(* IEC 61131-3 sources: axftcmlib/src/Axis/PosAxis, 6 files *)

(* ---- itfPosAxis.st ---- *)
USING Simatic.Ax.Commands;

NAMESPACE Simatic.Ax.axftcmlib.Motion

    INTERFACE itfPosAxis EXTENDS itfSpeedAxis

    METHOD MoveAbsolute  : itfCommand
        VAR_INPUT
            Position : LREAL; // Absolute target position
            Velocity : LReal := 100.0;
        END_VAR
    END_METHOD

    METHOD MoveRelative  : itfCommand
        VAR_INPUT
            Distance : LREAL; // Distance for the positioning process (negative or positive)
            Velocity : LReal := 100.0;
        END_VAR
    END_METHOD

    METHOD HomeDirect  : itfCommand
        VAR_INPUT
            Position : LREAL; // Distance for the positioning process (negative or positive)
        END_VAR
    END_METHOD

END_INTERFACE

END_NAMESPACE

(* ---- commandActiveHoming.st ---- *)
USING Simatic.Ax.IO.Input;
USING Simatic.Ax.IO.Input;
USING Simatic.Ax.Commands;
USING Simatic.Ax.IO.Input;

NAMESPACE Simatic.Ax.axftcmlib.Motion

    CLASS INTERNAL commandActiveHoming
        EXTENDS ExecuteCommand
        VAR
            _AxisRef : REF_TO TO_PosAxis;
            _velocity : LREAL;
            _direction : Direction;
            _position : LREAL;
            _iRefSensor : ItfBinSignal;
            _exec : BOOL;
        END_VAR

        METHOD PUBLIC Start : itfCommand
            VAR_INPUT
                AxisRef : REF_TO TO_PosAxis;
                Velocity : LREAL := 100.0;
                Direction : Direction;
                Position : LREAL := 0.0;
                RefSensor : ItfBinSignal;
            END_VAR
            _AxisRef := AxisRef;
            _velocity := Velocity;
            _direction := Direction;
            _position := Position;
            _iRefSensor := RefSensor;
            THIS.ExecuteWithRisingEdge();
            Start := THIS;
        END_METHOD

        METHOD PROTECTED OVERRIDE Execute
            IF NOT (_exec) THEN
                RETURN;
            END_IF;
            IF (NOT _AxisRef^.IsPoweredOn()) THEN
                THIS.SetError(WORD#16#8001);
            ELSE
                _AxisRef^.Run(TRUE);
                IF (_iRefSensor.QRis()) THEN
                    _AxisRef^.Run(FALSE);
                    _Done := _AxisRef^.SetPosition(value := _position);
                    ;
                END_IF;
            END_IF;
        END_METHOD

        METHOD PROTECTED OVERRIDE SetExecute
            VAR_INPUT
                exec : BOOL;
            END_VAR
            _exec := exec;
            IF (exec) THEN
                THIS.InitState();
                IF (_AxisRef = NULL) THEN
                    THIS.SetError(WORD#16#8003);
                    RETURN;
                ELSIF (_iRefSensor = NULL) THEN
                    THIS.SetError(WORD#16#8004);
                    RETURN;
                END_IF;
                IF (NOT _AxisRef^.IsPoweredOn()) THEN
                    THIS.SetError(WORD#16#8001);
                ELSIF (_AxisRef^.IsRunning()) THEN
                    THIS.SetError(WORD#16#8002); // Can not be homed because axis is not stillstanding
                END_IF;
            END_IF;
        END_METHOD
    END_CLASS

END_NAMESPACE

(* ---- commandHomeDirect.st ---- *)
USING Simatic.Ax.Commands;

NAMESPACE Simatic.Ax.axftcmlib.Motion

    CLASS INTERNAL commandHomeDirect
        EXTENDS ExecuteCommand
        VAR
            _AxisRef : REF_TO TO_PosAxis;
            _position : LReal;
        END_VAR

        METHOD PUBLIC Start : itfCommand
            VAR_INPUT
                AxisRef : REF_TO TO_PosAxis;
                Position : LREAL := 0.0;
            END_VAR
            _AxisRef := AxisRef;
            _position := Position;
            THIS.ExecuteWithRisingEdge();
            Start := THIS;
        END_METHOD

        METHOD PROTECTED OVERRIDE Execute
            IF (NOT _AxisRef^.isPowerdOn) THEN
                THIS.SetError(WORD#16#8001);
            ELSE
                ;
            END_IF;
        END_METHOD

        METHOD PROTECTED OVERRIDE SetExecute
            VAR_INPUT
                exec : BOOL;
            END_VAR
            IF (NOT _AxisRef^.isPowerdOn) THEN
                THIS.SetError(WORD#16#8001);
            ELSIF (_AxisRef^.IsRunning()) THEN
                THIS.SetError(WORD#16#8002);  // Con not be homed because axis is not stillstanding
            ELSE
                _Done := _AxisRef^.SetPosition(value := _position);
            END_IF;

        END_METHOD
    END_CLASS

END_NAMESPACE

(* ---- commandMoveAbsolute.st ---- *)
USING Simatic.Ax.Commands;

NAMESPACE Simatic.Ax.axftcmlib.Motion

    CLASS INTERNAL commandMoveAbsolute
        EXTENDS ExecuteCommand
        VAR
            _AxisRef : REF_TO TO_PosAxis;
            _velocity : LREAL;
            _position : LREAL;
        END_VAR
        VAR PRIVATE
            _execute : BOOL;
        END_VAR

        METHOD PUBLIC Start : itfCommand
            VAR_INPUT
                AxisRef : REF_TO TO_PosAxis;
                Velocity : LREAL := LREAL#100.0;
                Position : LREAL := 0.0;
            END_VAR
            _AxisRef := AxisRef;
            _velocity := Velocity;
            _position := Position;
            // Determine Direction
            IF (_position < THIS._AxisRef^.GetPosition()) THEN
                _AxisRef^.Direction := Direction#NegativeDirection;
            ELSIF (_position > THIS._AxisRef^.GetPosition()) THEN
                _AxisRef^.Direction := Direction#PositiveDirection;
            ELSE // distance = 0 --> do nothing
                THIS.SetDone();
                RETURN;
            END_IF;
            THIS.ExecuteWithRisingEdge();
            Start := THIS;
        END_METHOD

        METHOD PROTECTED OVERRIDE Execute
            VAR_TEMP
                _x : LREAL;
            END_VAR
            IF NOT (_execute) THEN
                THIS._Done := FALSE;
                THIS._Error := FALSE;
                RETURN;
            END_IF;

            // Axis must be powerd on and homed
            IF (NOT _AxisRef^.IsPoweredOn()) THEN
                THIS.SetError(WORD#16#8001);
                RETURN;
            ELSIF (NOT _AxisRef^.IsHomed()) THEN
                THIS.SetError(WORD#16#8003);
                RETURN;
            END_IF;
            _AxisRef^.Velocity := _velocity;
            _AxisRef^.Run(TRUE);
            _x := _AxisRef^.GetPosition();
            IF (_AxisRef^.Direction = Direction#NegativeDirection) THEN
                IF (_AxisRef^.GetPosition() <= _position) THEN
                    THIS.SetDone();
                    _AxisRef^.Run(FALSE);
                END_IF;
            ELSE
                IF (_AxisRef^.GetPosition() >= _position) THEN
                    THIS.SetDone();
                    _AxisRef^.Run(FALSE);
                END_IF;
            END_IF;
        END_METHOD

        METHOD PROTECTED OVERRIDE SetExecute
            VAR_INPUT
                exec : BOOL;
            END_VAR
            _execute := exec;
        END_METHOD
    END_CLASS

END_NAMESPACE

(* ---- commandMoveRelative.st ---- *)
USING Simatic.Ax.Commands;

NAMESPACE Simatic.Ax.axftcmlib.Motion

    CLASS INTERNAL commandMoveRelative
        EXTENDS ExecuteCommand
        VAR
            _AxisRef : REF_TO TO_PosAxis;
            _velocity : LREAL;
            _distance : LREAL;
        END_VAR
        VAR PRIVATE
            _execute : BOOL;
        END_VAR

        METHOD PUBLIC Start : itfCommand
            VAR_INPUT
                AxisRef : REF_TO TO_PosAxis;
                Velocity : LREAL := LREAL#100.0;
                Distance : LREAL := 0.0;
            END_VAR
            THIS._Done := FALSE;
            THIS._Error := FALSE;
            _AxisRef := AxisRef;
            _velocity := Velocity;
            _distance := Distance;
            _AxisRef^.Encoder.ResetRelative(); // Reset Reletive postioning counter
            // Determine Direction
            IF (_distance < 0.0) THEN
                _AxisRef^.Direction := Direction#NegativeDirection;
            ELSIF (_distance > 0.0) THEN
                _AxisRef^.Direction := Direction#PositiveDirection;
            ELSE // distance = 0 --> do nothing
                THIS.SetDone();
                Start := THIS;
                RETURN;
            END_IF;
            THIS.ExecuteWithRisingEdge();
            Start := THIS;
            _AxisRef^.Encoder.ResetRelative();
        END_METHOD

        METHOD PROTECTED OVERRIDE Execute
            VAR_TEMP
                _x : LREAL;
            END_VAR
            IF NOT (_execute) THEN
                RETURN;
            END_IF;
            // Axis must be powerd on and homed
            IF (NOT _AxisRef^.IsPoweredOn()) THEN
                THIS.SetError(WORD#16#8001);
                RETURN;
            ELSIF (NOT _AxisRef^.IsHomed()) THEN
                THIS.SetError(WORD#16#8003);
                RETURN;
            END_IF;
            _AxisRef^.Velocity := _velocity;
            _AxisRef^.Run(TRUE);
            _x := _AxisRef^.GetRelativePosition();
            IF (_AxisRef^.Direction = Direction#NegativeDirection) THEN
                IF (_AxisRef^.GetRelativePosition() <= _distance) THEN
                    THIS.SetDone();
                    _AxisRef^.Run(FALSE);
                END_IF;
            ELSE
                IF (_AxisRef^.GetRelativePosition() >= _distance) THEN
                    THIS.SetDone();
                    _AxisRef^.Run(FALSE);
                END_IF;
            END_IF;
        END_METHOD

        METHOD PROTECTED OVERRIDE SetExecute
            VAR_INPUT
                exec : BOOL;
            END_VAR
            _execute := exec;
        END_METHOD
    END_CLASS

END_NAMESPACE

(* ---- PosAxis.st ---- *)
USING Simatic.Ax.IO.Input;
USING Simatic.Ax.Commands;

NAMESPACE Simatic.Ax.axftcmlib.Motion

    CLASS PosAxis
        EXTENDS PosAxisImpl

        METHOD PUBLIC Attach : BOOL
            VAR_INPUT
                axis : REF_TO TO_PosAxis;
            END_VAR
            ;
            _PosAxisRef := axis;
            _SpeedAxisRef := axis;
            SUPER.Attach(axis);
            Attach := THIS.IsAttached();
        END_METHOD
    END_CLASS

    CLASS INTERNAL PosAxisImpl
        EXTENDS SpeedAxisImpl
        IMPLEMENTS itfPosAxis
        VAR PROTECTED
            _PosAxisRef : REF_TO TO_PosAxis;
            _commandMoveRelative : commandMoveRelative;
            _commandMoveAbsolute : commandMoveAbsolute;
            _commandHomeDirect : commandHomeDirect;
            _commandActiveHoming : commandActiveHoming;
        END_VAR

        METHOD PROTECTED OVERRIDE MakeAxisAbstract
            ;
        END_METHOD

        METHOD PUBLIC MoveAbsolute : itfCommand
            VAR_INPUT
                Position : LREAL;
                Velocity : LREAL := 100.0;
            END_VAR
            MoveAbsolute := _commandMoveAbsolute.Start(AxisRef := _PosAxisRef, Position := Position, Velocity := Velocity);
            ;
        END_METHOD

        METHOD PUBLIC MoveRelative : itfCommand
            VAR_INPUT
                Distance : LREAL := 0.0;
                Velocity : LREAL := 100.0;
            END_VAR
            MoveRelative := _commandMoveRelative.Start(AxisRef := _PosAxisRef, Distance := Distance, Velocity := Velocity);
            ;
        END_METHOD

        METHOD PUBLIC HomeDirect : itfCommand
            VAR_INPUT
                Position : LREAL;
            END_VAR
            HomeDirect := _commandHomeDirect.Start(AxisRef := _PosAxisRef, Position := Position);
        END_METHOD

        METHOD PUBLIC ActiveHoming : itfCommand
            VAR_INPUT
                Position : LREAL;
                Direction : Direction;
                RefSensor : ItfBinSignal;
            END_VAR
            ActiveHoming := _commandActiveHoming.Start(AxisRef := _PosAxisRef, Direction := Direction, Position := Position, RefSensor := RefSensor);
        END_METHOD
    END_CLASS

END_NAMESPACE
